(*
SPDX-FileCopyrightText: © 2026 Oleksandr Tiutyk <trofimich@gmail.com>
SPDX-License-Identifier: MIT
License: https://opensource.org/license/mit
*)

(*!
<summary>
Base automation component that coordinates children and routes requests through the component hierarchy.
</summary>
<description>
Action permissions are checked locally and then through parents, stopping at the first rejection. A missing
local policy permits that level; permission is granted only if no level rejects the request. Indexed Try
lookups return borrowed interfaces or null and do not propagate exceptions. Initialization validates required
dependencies before hooks. Each fixed child slot must identify a distinct child whose Parent is this branch.
Cycle-service hooks remain available while disabled in WORKING or STOPPED;
state changes end obsolete child phases. Use one owner task without recursive Execute.
</description>
*)

FUNCTION_BLOCK ABSTRACT BranchAutomationComponent EXTENDS AutomationComponent IMPLEMENTS IParentAutomationComponent
VAR
	{attribute 'hide'} 
	_ActionPermissionPolicy : TOF_Core.IActionPermissionPolicy;
	
	{attribute 'hide'} 
	_ChildCriticalErrorHandlingPolicy : IChildCriticalErrorHandlingPolicy;

	_ChildHierarchyValidated : BOOL;
END_VAR

{attribute 'monitoring' := 'call'}
PROPERTY FINAL ActionPermissionPolicy : TOF_Core.IActionPermissionPolicy
GET
ActionPermissionPolicy := _ActionPermissionPolicy;
END_GET
SET
_ActionPermissionPolicy := ActionPermissionPolicy;
END_SET
END_PROPERTY

METHOD FINAL BroadcastEvent
VAR_INPUT
	event : TOF_Core.IEvent;
END_VAR
VAR
	stopPropagation : BOOL;
	
	i : TOF_Core.INT_INDEX;
	
	child : IChildAutomationComponent;
	childAsBroadcastEventDispatcher : TOF_Core.IBroadcastEventDispatcher;
END_VAR
OnEventReceived(event := event, stopPropagation => stopPropagation);

IF stopPropagation THEN
	RETURN;
END_IF

FOR i := 0 TO ChildCount - 1 DO
	child := TryGetChildByIndex(index := i);
	
	IF child = 0 OR_ELSE NOT __QUERYINTERFACE(child, childAsBroadcastEventDispatcher) THEN
		CONTINUE;
	END_IF
	
	childAsBroadcastEventDispatcher.BroadcastEvent(event := event);
END_FOR
END_METHOD

{attribute 'monitoring' := 'call'}
PROPERTY ABSTRACT ChildCount : TOF_Core.INT_LENGTH
GET
END_GET
END_PROPERTY

{attribute 'monitoring' := 'call'}
PROPERTY FINAL ChildCriticalErrorHandlingPolicy : IChildCriticalErrorHandlingPolicy
GET
ChildCriticalErrorHandlingPolicy := _ChildCriticalErrorHandlingPolicy;
END_GET
SET
_ChildCriticalErrorHandlingPolicy := ChildCriticalErrorHandlingPolicy;
END_SET
END_PROPERTY

(*!
<summary>Disables the branch, its children and invokes disable hooks.</summary>
<description>
Hook or child exceptions propagate to the caller without rolling back already disabled children.
</description>
*)
METHOD FINAL Disable
VAR
	i : INT;
	
	child : IChildAutomationComponent;

	exceptionCode : __SYSTEM.ExceptionCode;
END_VAR
VAR_INST
	disabling : BOOL;
END_VAR
IF NOT _Enabled OR_ELSE disabling THEN
	RETURN;
END_IF

disabling := TRUE;

__TRY
	OnBeforeChildrenDisable();
	
	FOR i := 0 TO ChildCount - 1 DO
		child := TryGetChildByIndex(index := i);
		
		IF child <> 0 THEN
			child.Disable();
		END_IF
	END_FOR
	
	OnAfterChildrenDisable();
	
	_Enabled := FALSE;
	
	disabling := FALSE;	
__CATCH(exceptionCode)
	disabling := FALSE;
	
	TOF_Core.ExceptionManager.ReThrowLastException(
		exceptionCode := exceptionCode,
		catchPointNamespaceName := NamespaceName,
		catchPointPOUName := __POUNAME(),
		catchPointPosition := __POSITION()
	);
__ENDTRY
END_METHOD

(*!
<summary>Advances stopped children while the branch remains enabled and stopped.</summary>
<description>
OnBeforeChildrenStopped may call Reset. A state or enablement change ends this phase before remaining
children or the after-stopped hook. Completed effects remain. Hook failures are logged; other failures may escape.
</description>
*)
METHOD PRIVATE FINAL doStop
VAR
	exceptionCode : __SYSTEM.ExceptionCode;
	exception : TOF_Core.IException;	
	exceptionReaction : TOF_Core.EXCEPTION_REACTION;

	i : INT;
	
	child : IChildAutomationComponent;
END_VAR
__TRY
	OnBeforeChildrenStopped();
__CATCH(exceptionCode)
	exception := TOF_Core.ExceptionManager.GetLastException(
		exceptionCode := exceptionCode,
		catchPointNamespaceName := NamespaceName,
		catchPointPOUName := __POUNAME(),
		catchPointPosition := __POSITION()
	);	

	exceptionReaction := OnHandleException(exception := exception, failedMethodName := 'OnBeforeChildrenStopped');

	TOF_Core.LogManager.TryLogException(
		exception := exception,
		severity := GetErrorSeverityByExceptionReaction(exceptionReaction := exceptionReaction),
		topic1 := "AutomationComponent",
		topic2 := "AutomationComponent.OnBeforeChildrenStopped"
	);
__ENDTRY	

IF NOT Enabled OR_ELSE _OperationalState <> OPERATIONAL_STATE.STOPPED THEN
	RETURN;
END_IF

FOR i := 0 TO ChildCount - 1 DO
	child := TryGetChildByIndex(index := i);
	
	IF child = 0 OR_ELSE NOT child.Enabled THEN
		CONTINUE;
	END_IF
	
	CASE child.OperationalState OF
		OPERATIONAL_STATE.WORKING:			
			child.Stop(reason := TOF_Core.WideStrings.Concat255("Parent device (", Name, ") stopped"));
		
		OPERATIONAL_STATE.STOPPED:
			child.Execute();
	END_CASE

	IF NOT Enabled OR_ELSE _OperationalState <> OPERATIONAL_STATE.STOPPED THEN
		RETURN;
	END_IF
END_FOR

__TRY
	OnAfterChildrenStopped();
__CATCH(exceptionCode)
	exception := TOF_Core.ExceptionManager.GetLastException(
		exceptionCode := exceptionCode,
		catchPointNamespaceName := NamespaceName,
		catchPointPOUName := __POUNAME(),
		catchPointPosition := __POSITION()
	);	

	exceptionReaction := OnHandleException(exception := exception, failedMethodName := 'OnAfterChildrenStopped');

	TOF_Core.LogManager.TryLogException(
		exception := exception,
		severity := GetErrorSeverityByExceptionReaction(exceptionReaction := exceptionReaction),
		topic1 := "AutomationComponent",
		topic2 := "AutomationComponent.OnAfterChildrenStopped"
	);
__ENDTRY
END_METHOD

(*!
<summary>Advances children according to the selected critical-error reaction.</summary>
<description>
Ignore and continue preserve traversal of later children and the after-working hook. Stop ends traversal.
A non-critical error copied from a faulted child under SET_ERROR_AND_CONTINUE is retained without calling
OnRecover while any enabled child still holds a critical error handled with continue. An exception raised by
OnRecover always records a copied CRITICAL error and stops the branch without consulting
ExceptionHandlingPolicy. State or enablement changes end the obsolete phase; completed effects remain.
</description>
*)
METHOD PRIVATE doWork
VAR
	exceptionCode : __SYSTEM.ExceptionCode;
	exception : TOF_Core.IException;	
	exceptionReaction : TOF_Core.EXCEPTION_REACTION;

	childCriticalErrorReaction : CHILD_CRITICAL_ERROR_REACTION;

	i : INT;
	
	child : IChildAutomationComponent;
END_VAR
// automatic non-critical error recovering
IF _OperationalState = OPERATIONAL_STATE.WORKING
	AND_THEN HasError
	AND_THEN _Error.Severity <> TOF_Core.ERROR_SEVERITY.CRITICAL
	AND_THEN NOT hasActiveChildCriticalError()
THEN
	_Error.Clear();
	
	__TRY
		OnRecover();
	__CATCH(exceptionCode)		
		exception := TOF_Core.ExceptionManager.GetLastException(
			exceptionCode := exceptionCode,
			catchPointNamespaceName := NamespaceName,
			catchPointPOUName := __POUNAME(),
			catchPointPosition := __POSITION()
		);

		// An OnRecover failure always stops the branch with a critical error without consulting the policy.
		ProcessException(
			exception := exception,
			exceptionReaction := TOF_Core.EXCEPTION_REACTION.SET_ERROR_AND_STOP,
			exceptionSourceHint := "OnRecover error"
		);

		RETURN;
	__ENDTRY
END_IF

IF NOT Enabled OR_ELSE _OperationalState <> OPERATIONAL_STATE.WORKING THEN
	RETURN;
END_IF

__TRY
	OnBeforeChildrenWorking();
__CATCH(exceptionCode)
	exception := TOF_Core.ExceptionManager.GetLastException(
		exceptionCode := exceptionCode,
		catchPointNamespaceName := NamespaceName,
		catchPointPOUName := __POUNAME(),
		catchPointPosition := __POSITION()
	);	

	exceptionReaction := OnHandleException(exception := exception, failedMethodName := 'OnBeforeChildrenWorking');

	ProcessException(
		exception := exception,
		exceptionReaction := exceptionReaction,
		exceptionSourceHint := "OnBeforeChildrenWorking error"
	);

	IF exceptionReaction = TOF_Core.EXCEPTION_REACTION.SET_ERROR_AND_STOP THEN
		RETURN;		
	END_IF
__ENDTRY	

IF NOT Enabled OR_ELSE _OperationalState <> OPERATIONAL_STATE.WORKING THEN
	RETURN;
END_IF

FOR i := 0 TO ChildCount - 1 DO
	child := TryGetChildByIndex(index := i);
	
	IF child <> 0
		AND_THEN child.Enabled
		AND_THEN (
			child.OperationalState = OPERATIONAL_STATE.WORKING
			OR_ELSE child.OperationalState = OPERATIONAL_STATE.STOPPED
		)
	THEN
		child.Execute();
		
		IF child.HasError AND_THEN child.Error.Severity = TOF_Core.ERROR_SEVERITY.CRITICAL THEN
			childCriticalErrorReaction := HandleChildCriticalError(childWithError := child);
			
			ProcessChildError(
				childError := child.Error,
				childErrorReaction := childCriticalErrorReaction,
				childErrorSourceHint := TOF_Core.WideStrings.Concat255("Child[", TO_WSTRING(i), "](", child.Name, ").Execute error")
			);
			
			IF childCriticalErrorReaction = CHILD_CRITICAL_ERROR_REACTION.SET_ERROR_AND_STOP THEN
				RETURN;
			END_IF
		END_IF
	END_IF

	IF NOT Enabled OR_ELSE _OperationalState <> OPERATIONAL_STATE.WORKING THEN
		RETURN;
	END_IF
END_FOR

__TRY
	OnAfterChildrenWorking();
__CATCH(exceptionCode)
	exception := TOF_Core.ExceptionManager.GetLastException(
		exceptionCode := exceptionCode,
		catchPointNamespaceName := NamespaceName,
		catchPointPOUName := __POUNAME(),
		catchPointPosition := __POSITION()
	);	

	exceptionReaction := OnHandleException(exception := exception, failedMethodName := 'OnAfterChildrenWorking');

	ProcessException(
		exception := exception,
		exceptionReaction := exceptionReaction,
		exceptionSourceHint := "OnAfterChildrenWorking error"
	);

	IF exceptionReaction = TOF_Core.EXCEPTION_REACTION.SET_ERROR_AND_STOP THEN
		RETURN;		
	END_IF
__ENDTRY
END_METHOD

(*!
<summary>Enables the branch, optionally its children, and invokes enable hooks.</summary>
<description>
Enabling does not automatically reset a STOPPED branch or STOPPED children; they remain STOPPED after
Enable until explicitly Reset. If this branch has a disabled parent, enables the parent with
includeChildren := FALSE.
</description>
<param name="includeChildren">When TRUE, recursively enables child components.</param>
*)
METHOD FINAL Enable
VAR_INPUT
	includeChildren : BOOL := TRUE;
END_VAR
VAR
	i : INT;
	
	child : IChildAutomationComponent;

	exceptionCode : __SYSTEM.ExceptionCode;
	
	thisAsChildAutomationComponent : IChildAutomationComponent;
	parent : IParentAutomationComponent;
END_VAR
VAR_INST
	enabling : BOOL;
END_VAR
IF _Enabled OR_ELSE enabling THEN
	RETURN;
END_IF

enabling := TRUE;

__TRY
	OnBeforeChildrenEnable();
	
	IF includeChildren THEN
		FOR i := 0 TO ChildCount - 1 DO
			child := TryGetChildByIndex(index := i);
			
			IF child <> 0 THEN
				child.Enable(includeChildren := includeChildren);
			END_IF
		END_FOR	
	END_IF
	
	OnAfterChildrenEnable();
	
	IF __QUERYINTERFACE(THIS^, thisAsChildAutomationComponent) THEN
		parent := thisAsChildAutomationComponent.Parent;

		IF parent <> 0 AND_THEN NOT parent.Enabled THEN
			parent.Enable(includeChildren := FALSE);
		END_IF
	END_IF
	
	_Enabled := TRUE;
	
	enabling := FALSE;
__CATCH(exceptionCode)
	enabling := FALSE;
	
	TOF_Core.ExceptionManager.ReThrowLastException(
		exceptionCode := exceptionCode,
		catchPointNamespaceName := NamespaceName,
		catchPointPOUName := __POUNAME(),
		catchPointPosition := __POSITION()
	);
__ENDTRY
END_METHOD

(*!
<summary>Services an initialized branch and advances its enabled execution phases.</summary>
<description>
Only WORKING and STOPPED are serviced. Cycle-service hooks run even while disabled, before and after
enabled input, working or stopped, and output phases. They may enable, disable, stop or reset the branch;
enablement is checked again before work and output. INITIALIZING and INVALID do nothing. The final service
hook also follows handled stop reactions; an escaping nested failure may abort the call. Use one owner task
without recursive Execute. Completed callback effects are not rolled back.
</description>
*)
{attribute 'estimated-stack-usage' := '99'}
METHOD FINAL Execute
VAR
	exceptionCode : __SYSTEM.ExceptionCode;
	exception : TOF_Core.IException;
	exceptionReaction : TOF_Core.EXCEPTION_REACTION;
	runEnabledPhases : BOOL;
END_VAR
IF _OperationalState <> OPERATIONAL_STATE.WORKING
	AND_THEN _OperationalState <> OPERATIONAL_STATE.STOPPED
THEN
	RETURN;
END_IF

runEnabledPhases := TRUE;

__TRY
	OnCycleStart();
__CATCH(exceptionCode)
	exception := TOF_Core.ExceptionManager.GetLastException(
		exceptionCode := exceptionCode,
		catchPointNamespaceName := NamespaceName,
		catchPointPOUName := __POUNAME(),
		catchPointPosition := __POSITION()
	);
	exceptionReaction := OnHandleException(exception := exception, failedMethodName := 'OnCycleStart');

	ProcessException(
		exception := exception,
		exceptionReaction := exceptionReaction,
		exceptionSourceHint := "OnCycleStart error"
	);

	IF exceptionReaction = TOF_Core.EXCEPTION_REACTION.SET_ERROR_AND_STOP THEN
		runEnabledPhases := FALSE;
	END_IF
__ENDTRY

IF runEnabledPhases AND_THEN Enabled THEN
	__TRY
		OnBeforeExecute();
	__CATCH(exceptionCode)
		exception := TOF_Core.ExceptionManager.GetLastException(
			exceptionCode := exceptionCode,
			catchPointNamespaceName := NamespaceName,
			catchPointPOUName := __POUNAME(),
			catchPointPosition := __POSITION()
		);
		exceptionReaction := OnHandleException(exception := exception, failedMethodName := 'OnBeforeExecute');

		ProcessException(
			exception := exception,
			exceptionReaction := exceptionReaction,
			exceptionSourceHint := "OnBeforeExecute error"
		);

		IF exceptionReaction = TOF_Core.EXCEPTION_REACTION.SET_ERROR_AND_STOP THEN
			runEnabledPhases := FALSE;
		END_IF
	__ENDTRY

	IF runEnabledPhases AND_THEN Enabled THEN
		CASE _OperationalState OF
			OPERATIONAL_STATE.WORKING:
				doWork();

			OPERATIONAL_STATE.STOPPED:
				doStop();
		END_CASE
	END_IF

	IF runEnabledPhases AND_THEN Enabled THEN
		__TRY
			OnAfterExecute();
		__CATCH(exceptionCode)
			exception := TOF_Core.ExceptionManager.GetLastException(
				exceptionCode := exceptionCode,
				catchPointNamespaceName := NamespaceName,
				catchPointPOUName := __POUNAME(),
				catchPointPosition := __POSITION()
			);
			exceptionReaction := OnHandleException(exception := exception, failedMethodName := 'OnAfterExecute');

			ProcessException(
				exception := exception,
				exceptionReaction := exceptionReaction,
				exceptionSourceHint := "OnAfterExecute error"
			);
		__ENDTRY
	END_IF
END_IF

__TRY
	OnCycleEnd();
__CATCH(exceptionCode)
	exception := TOF_Core.ExceptionManager.GetLastException(
		exceptionCode := exceptionCode,
		catchPointNamespaceName := NamespaceName,
		catchPointPOUName := __POUNAME(),
		catchPointPosition := __POSITION()
	);
	exceptionReaction := OnHandleException(exception := exception, failedMethodName := 'OnCycleEnd');

	ProcessException(
		exception := exception,
		exceptionReaction := exceptionReaction,
		exceptionSourceHint := "OnCycleEnd error"
	);
__ENDTRY
END_METHOD

METHOD GetEffectiveChildCriticalErrorHandlingPolicy : IChildCriticalErrorHandlingPolicy
VAR
	thisAsChildAutomationComponent : IChildAutomationComponent;
	parent : IParentAutomationComponent;
END_VAR
IF _ChildCriticalErrorHandlingPolicy <> 0 THEN
	GetEffectiveChildCriticalErrorHandlingPolicy := _ChildCriticalErrorHandlingPolicy;
ELSIF __QUERYINTERFACE(THIS^, thisAsChildAutomationComponent) THEN
	parent := thisAsChildAutomationComponent.Parent;

	IF parent <> 0 THEN
		GetEffectiveChildCriticalErrorHandlingPolicy := parent.GetEffectiveChildCriticalErrorHandlingPolicy();
	END_IF
END_IF
END_METHOD

METHOD PROTECTED FINAL HandleChildCriticalError : CHILD_CRITICAL_ERROR_REACTION
VAR_INPUT
	childWithError : IChildAutomationComponent;
END_VAR
VAR
	effectiveChildCriticalErrorHandlingPolicy : IChildCriticalErrorHandlingPolicy;
END_VAR
effectiveChildCriticalErrorHandlingPolicy := GetEffectiveChildCriticalErrorHandlingPolicy();

IF effectiveChildCriticalErrorHandlingPolicy <> 0 THEN
	HandleChildCriticalError := effectiveChildCriticalErrorHandlingPolicy.HandleChildCriticalError(
		childWithError := childWithError,
		handlingObject := THIS^
	);
ELSE
	HandleChildCriticalError := CHILD_CRITICAL_ERROR_REACTION.SET_ERROR_AND_STOP;
END_IF
END_METHOD

(*!
<summary>Checks whether any enabled child still holds a critical error handled with continue.</summary>
<description>
Prevents premature automatic non-critical error clearing and OnRecover calls while an enabled child
remains faulted with a critical error under SET_ERROR_AND_CONTINUE.
</description>
*)
METHOD PRIVATE hasActiveChildCriticalError : BOOL
VAR
	i : INT;
	child : IChildAutomationComponent;
	childCriticalErrorReaction : CHILD_CRITICAL_ERROR_REACTION;
END_VAR
FOR i := 0 TO ChildCount - 1 DO
	child := TryGetChildByIndex(index := i);

	IF child <> 0
		AND_THEN child.Enabled
		AND_THEN child.HasError
		AND_THEN child.Error.Severity = TOF_Core.ERROR_SEVERITY.CRITICAL
	THEN
		childCriticalErrorReaction := HandleChildCriticalError(childWithError := child);

		IF childCriticalErrorReaction = CHILD_CRITICAL_ERROR_REACTION.SET_ERROR_AND_CONTINUE THEN
			hasActiveChildCriticalError := TRUE;

			RETURN;
		END_IF
	END_IF
END_FOR
END_METHOD

(*!
<summary>Validates required dependencies and advances branch initialization.</summary>
<description>
Required storage and child slots are checked before initialization hooks. Empty compositions are valid.
Before the first initialization hook, each child must name this branch as Parent and appear in exactly one slot.
Keep the composition stable thereafter. A mismatch or duplicate records a critical error and makes the branch INVALID.
An INVALID child immediately makes this branch INVALID and copies its error when available.
During initialization, the branch expands its effective initialization timeout to at least the maximum
InitializationTimeout of its children. OnAfterChildrenInitializing runs only once all children have completed
initialization. FALSE reports pending work or failure. Caught initialization failures return FALSE and record
a critical error in terminal INVALID. TRUE reports completed initialization, including an already stopped
component. Callback effects are not rolled back. Child types require a live constructor-bound parent.
</description>
*)
METHOD FINAL Initialize : BOOL
VAR
	i : INT;
	previousIndex : INT;
	expectedParent : IParentAutomationComponent;
	childParent : IParentAutomationComponent;
	hierarchyError : WSTRING(255);
		
	child : IChildAutomationComponent;
	previousChild : IChildAutomationComponent;
	childInitialized : BOOL;
	
	exceptionCode : __SYSTEM.ExceptionCode;
	exception : TOF_Core.IException;
	
END_VAR
IF _OperationalState <> OPERATIONAL_STATE.INITIALIZING THEN
	Initialize := _OperationalState <> OPERATIONAL_STATE.INVALID;

	RETURN;
END_IF

__TRY
	Validate();
	expectedParent := THIS^;

	FOR i := 0 TO ChildCount - 1 DO
		child := TryGetChildByIndex(index := i);

		IF child = 0 THEN
			TOF_Core.Exceptions.ThrowDataMemberNotSpecified(
				sourceNamespaceName := NamespaceName,
				sourceClassName := ClassName,
				sourcePOUName := __POUNAME(),
				sourcePosition := __POSITION(),
				dataMemberName := TOF_Core.Strings.Concat255('Child[', TO_STRING(i), ']')
			);			
		END_IF

		IF _ChildHierarchyValidated THEN
			CONTINUE;
		END_IF

		childParent := child.Parent;

		IF childParent <> expectedParent THEN
			hierarchyError := TOF_Core.WideStrings.Concat255(
				Name,
				": Children[",
				TO_WSTRING(i),
				"] (",
				child.Name,
				") has a different Parent"
			);
		ELSE
			FOR previousIndex := 0 TO i - 1 DO
				previousChild := TryGetChildByIndex(index := previousIndex);

				IF previousChild = child THEN
					hierarchyError := TOF_Core.WideStrings.Concat255(
						Name,
						": Children[",
						TO_WSTRING(i),
						"] (",
						child.Name,
						") duplicates Children[",
						TO_WSTRING(previousIndex),
						"]"
					);

					EXIT;
				END_IF
			END_FOR
		END_IF

		IF hierarchyError <> "" THEN
			TOF_Core.Exceptions.ThrowClassInitialization(
				sourceNamespaceName := NamespaceName,
				sourceClassName := ClassName,
				sourcePOUName := __POUNAME(),
				sourcePosition := __POSITION(),
				errorMessage := hierarchyError
			);
		END_IF
	END_FOR

	_ChildHierarchyValidated := TRUE;
	OnBeforeChildrenInitializing();

	IF _InitializationTimer.PT = T#0S THEN
		_InitializationTimer.PT := Parameters.InitializationTimeout;
	END_IF

	Initialize := TRUE;

	FOR i := 0 TO ChildCount - 1 DO
		child := TryGetChildByIndex(index := i);

		IF child = 0 THEN
			TOF_Core.Exceptions.ThrowDataMemberNotSpecified(
				sourceNamespaceName := NamespaceName,
				sourceClassName := ClassName,
				sourcePOUName := __POUNAME(),
				sourcePosition := __POSITION(),
				dataMemberName := TOF_Core.Strings.Concat255('Child[', TO_STRING(i), ']')
			);
		END_IF

		childInitialized := child.Initialize();

		IF child.OperationalState = OPERATIONAL_STATE.INVALID THEN
			Initialize := FALSE;

			IF child.HasError THEN
				_Error := child.Error;
				_Error.SetSeverity(severity := TOF_Core.ERROR_SEVERITY.CRITICAL);
				SetOperationalState(
					state := OPERATIONAL_STATE.INVALID,
					reason := TOF_Core.WideStrings.Concat255("Child[", TO_WSTRING(i), "] initialization failed")
				);

				RETURN;
			END_IF

			TOF_Core.Exceptions.ThrowStandard(
				sourceNamespaceName := NamespaceName,
				sourceClassName := ClassName,
				sourcePOUName := __POUNAME(),
				sourcePosition := __POSITION(),
				message := "A child entered INVALID during initialization without an error diagnostic."
			);
		END_IF

		IF child.InitializationTimeout > _InitializationTimer.PT THEN
			_InitializationTimer.PT := child.InitializationTimeout;
		END_IF

		Initialize := Initialize AND childInitialized;
	END_FOR

	Initialize := Initialize AND_THEN OnAfterChildrenInitializing();
	
	IF Initialize THEN
		SetOperationalState(state := OPERATIONAL_STATE.WORKING, reason := "Successfull initialization");
	ELSE
		_InitializationTimer(IN := TRUE);
		
		IF _InitializationTimer.Q THEN		
			TOF_Core.Exceptions.ThrowTimeout(
				sourceNamespaceName := NamespaceName,
				sourceClassName := ClassName,
				sourcePOUName := __POUNAME(),
				sourcePosition := __POSITION(),
				timeoutValue := _InitializationTimer.PT,
				operationName := "Initialization"
			);
		END_IF		
	END_IF	
__CATCH(exceptionCode)
	Initialize := FALSE;

	IF hierarchyError = "" THEN
		hierarchyError := "Initialization error";
	END_IF

	exception := TOF_Core.ExceptionManager.GetLastException(
		exceptionCode := exceptionCode,
		catchPointNamespaceName := NamespaceName,
		catchPointPOUName := __POUNAME(),
		catchPointPosition := __POSITION()
	);
	
	ProcessException(
		exception := exception,
		exceptionReaction := TOF_Core.EXCEPTION_REACTION.SET_ERROR_AND_CONTINUE,
		exceptionSourceHint := hierarchyError
	);					
__ENDTRY
END_METHOD

METHOD PROTECTED OnAfterChildrenDisable
END_METHOD

METHOD PROTECTED OnAfterChildrenEnable
END_METHOD

(*!
<summary>Completes branch initialization after all children have finished initializing.</summary>
<description>
Invoked only once every child has completed initialization (returned TRUE from Initialize). Return FALSE to
keep the branch in INITIALIZING until a subsequent Initialize call returns TRUE.
</description>
*)
METHOD PROTECTED OnAfterChildrenInitializing : BOOL
OnAfterChildrenInitializing := TRUE;
END_METHOD

METHOD PROTECTED OnAfterChildrenProcessInput
END_METHOD

(*!
<summary>Runs after the branch completes an output pass without changing its operational state.</summary>
<description>Both working and stopped passes may complete. An interrupted pass skips this hook.</description>
*)
METHOD PROTECTED OnAfterChildrenProcessOutput
END_METHOD

METHOD PROTECTED OnAfterChildrenReset
END_METHOD

METHOD PROTECTED OnAfterChildrenStopped
END_METHOD

METHOD PROTECTED OnAfterChildrenWorking
END_METHOD

(*!
<summary>Completes enabled processing after the working or stopped phase.</summary>
<description>
Execute checks Enabled again before calling this hook. STOPPED branches remain eligible. A handled stop
reaction in OnCycleStart or OnBeforeExecute skips this hook. The base implementation does nothing.
Exceptions follow the branch exception policy.
</description>
*)
METHOD PROTECTED OnAfterExecute
END_METHOD

METHOD PROTECTED OnBeforeChildrenDisable
END_METHOD

METHOD PROTECTED OnBeforeChildrenEnable
END_METHOD

(*!
<summary>Runs before child initialization on each pending initialization cycle.</summary>
<description>
Invoked after branch dependencies and child hierarchy validation succeed. Exceptions transition the branch to
terminal INVALID.
</description>
*)
METHOD PROTECTED OnBeforeChildrenInitializing
END_METHOD

METHOD PROTECTED OnBeforeChildrenProcessInput
END_METHOD

METHOD PROTECTED OnBeforeChildrenProcessOutput
END_METHOD

METHOD PROTECTED OnBeforeChildrenReset
END_METHOD

(*!
<summary>Runs before stopped-child traversal.</summary>
<description>
May call Reset. A state or enablement change ends this stopped phase before remaining children
and the after-stopped hook. Do not recursively call Execute.
</description>
*)
METHOD PROTECTED OnBeforeChildrenStopped
END_METHOD

METHOD PROTECTED OnBeforeChildrenWorking
END_METHOD

(*!
<summary>Prepares an enabled branch for its working or stopped phase.</summary>
<description>
Execute calls this hook after OnCycleStart if the branch is enabled and the enabled phases may proceed.
Execute then checks Enabled again and selects the phase using the current operational state. The base
implementation does nothing. Exceptions follow the branch exception policy.
</description>
*)
METHOD PROTECTED OnBeforeExecute
END_METHOD

(*!
<summary>Services the branch after the enabled phases have run or been skipped.</summary>
<description>
Execute reaches this hook even while disabled and after a handled stop reaction. An escaping exception
can end Execute before this hook runs. The base implementation does nothing. Exceptions raised here follow
the branch exception policy.
</description>
*)
METHOD PROTECTED OnCycleEnd
END_METHOD

(*!
<summary>Services the branch before Execute checks Enabled.</summary>
<description>
Execute calls this hook in WORKING and STOPPED, including while disabled. An override can process commands
that enable or disable the branch for this call. The base implementation does nothing. Exceptions follow
the branch exception policy.
</description>
*)
METHOD PROTECTED OnCycleStart
END_METHOD

(*!
<summary>
Checks local permission and then requests permission from the parent, stopping at the first rejection.
</summary>
<description>
A missing local policy permits this level. The local policy receives this branch as evaluatingObject; the
original descriptor and requester are forwarded unchanged to the parent. Returns TRUE only if no level rejects
the request. On FALSE, rejectReason contains the rejecting level's reason; on TRUE it must be ignored.
Evaluation exceptions propagate to the caller without becoming ordinary rejections. Inputs must be non-null
and live. Arguments are borrowed only during this synchronous call, without ownership transfer.
</description>
*)

METHOD FINAL RequestActionPermission : BOOL
VAR_INPUT
	actionDescriptor : TOF_Core.INamed;
	requestingObject : TOF_Core.IObject;
END_VAR
VAR_IN_OUT
	rejectReason : WSTRING(255);
END_VAR
VAR
	thisAsChildAutomationComponent : IChildAutomationComponent;
	parent : IParentAutomationComponent;
END_VAR
IF _ActionPermissionPolicy <> 0 THEN 
	RequestActionPermission := _ActionPermissionPolicy.CheckActionPermission(
		actionDescriptor := actionDescriptor,
		requestingObject := requestingObject,
		evaluatingObject := THIS^,
		rejectReason := rejectReason
	);
ELSE
	RequestActionPermission := TRUE;
END_IF

IF RequestActionPermission
	AND_THEN __QUERYINTERFACE(THIS^, thisAsChildAutomationComponent)
THEN
	parent := thisAsChildAutomationComponent.Parent;

	IF parent <> 0 THEN
		RequestActionPermission := parent.RequestActionPermission(
			actionDescriptor := actionDescriptor,
			requestingObject := requestingObject,
			rejectReason := rejectReason
		);
	END_IF
END_IF
END_METHOD

(*!
<summary>Attempts to resume an enabled stopped branch and its enabled children.</summary>
<description>
Clears the previous branch error before reset hooks. Disabled children are skipped and remain STOPPED if
later enabled until explicitly Reset. A failure of the branch's own reset hook (OnBeforeChildrenReset or
OnAfterChildrenReset) always leaves the branch STOPPED with a copied CRITICAL error without consulting
ExceptionHandlingPolicy; later children are not reset after OnBeforeChildrenReset fails. Ignore and
continue allow later children to reset and the branch to enter WORKING even if a child remains stopped.
Continue copies that error at ERROR severity; ignore leaves it local. Stop leaves the branch STOPPED. Reset
may be called from a stopped-cycle hook, but reset hooks must not reenter Reset. State or enablement changes
end traversal; completed effects remain.
</description>
*)
METHOD FINAL Reset
VAR
	exceptionCode : __SYSTEM.ExceptionCode;
	exception : TOF_Core.IException;	
	
	childCriticalErrorReaction : CHILD_CRITICAL_ERROR_REACTION;
	
	i : INT;
		
	child : IChildAutomationComponent;	
END_VAR
IF NOT Enabled OR_ELSE _OperationalState <> OPERATIONAL_STATE.STOPPED THEN
	RETURN;
END_IF

_Error.Clear();

__TRY
	OnBeforeChildrenReset();
__CATCH(exceptionCode)		
	exception := TOF_Core.ExceptionManager.GetLastException(
		exceptionCode := exceptionCode,
		catchPointNamespaceName := NamespaceName,
		catchPointPOUName := __POUNAME(),
		catchPointPosition := __POSITION()
	);

	// A failed reset hook always keeps the branch STOPPED with a critical error; the policy is not consulted.
	ProcessException(
		exception := exception,
		exceptionReaction := TOF_Core.EXCEPTION_REACTION.SET_ERROR_AND_STOP,
		exceptionSourceHint := "OnBeforeChildrenReset error"
	);

	RETURN;
__ENDTRY

IF NOT Enabled OR_ELSE _OperationalState <> OPERATIONAL_STATE.STOPPED THEN
	RETURN;
END_IF

FOR i := 0 TO ChildCount - 1 DO
	child := TryGetChildByIndex(index := i);
	
	IF child <> 0 AND_THEN child.Enabled THEN
		child.Reset();
		
		IF child.HasError AND_THEN child.Error.Severity = TOF_Core.ERROR_SEVERITY.CRITICAL THEN
			childCriticalErrorReaction := HandleChildCriticalError(childWithError := child);
			
			ProcessChildError(
				childError := child.Error,
				childErrorReaction := childCriticalErrorReaction,
				childErrorSourceHint := TOF_Core.WideStrings.Concat255("Child[", TO_WSTRING(i), "](", child.Name, ").Reset error")
			);

			IF childCriticalErrorReaction = CHILD_CRITICAL_ERROR_REACTION.SET_ERROR_AND_STOP THEN
				RETURN;
			END_IF
		END_IF
	END_IF

	IF NOT Enabled OR_ELSE _OperationalState <> OPERATIONAL_STATE.STOPPED THEN
		RETURN;
	END_IF
END_FOR

__TRY
	OnAfterChildrenReset();
	
	IF Enabled AND_THEN _OperationalState = OPERATIONAL_STATE.STOPPED THEN
		SetOperationalState(state := OPERATIONAL_STATE.WORKING, reason := "Reset");
	END_IF
__CATCH(exceptionCode)		
	exception := TOF_Core.ExceptionManager.GetLastException(
		exceptionCode := exceptionCode,
		catchPointNamespaceName := NamespaceName,
		catchPointPOUName := __POUNAME(),
		catchPointPosition := __POSITION()
	);

	// A failed reset hook always keeps the branch STOPPED with a critical error; the policy is not consulted.
	ProcessException(
		exception := exception,
		exceptionReaction := TOF_Core.EXCEPTION_REACTION.SET_ERROR_AND_STOP,
		exceptionSourceHint := "OnAfterChildrenReset error"
	);
__ENDTRY
END_METHOD

(*!
<summary>Transitions a WORKING branch and all WORKING children to OPERATIONAL_STATE.STOPPED.</summary>
<description>
Stops the branch and all WORKING children regardless of Enabled. Child Stop failures are logged as critical.
</description>
<param name="reason">Descriptive reason stored in OperationalStateReason.</param>
*)
METHOD FINAL Stop
VAR_INPUT
	reason : WSTRING(255) := "External stop";
END_VAR
VAR
	exceptionCode : __SYSTEM.ExceptionCode;
	exception : TOF_Core.IException;	

	i : INT;
	
	child : IChildAutomationComponent;
END_VAR
IF _OperationalState <> OPERATIONAL_STATE.WORKING THEN
	RETURN;
END_IF

SetOperationalState(state := OPERATIONAL_STATE.STOPPED, reason := reason);

FOR i := 0 TO ChildCount - 1 DO
	__TRY
		child := TryGetChildByIndex(index := i); 
		
		IF child <> 0 AND_THEN child.OperationalState = OPERATIONAL_STATE.WORKING THEN		
			child.Stop(reason := TOF_Core.WideStrings.Concat255("Parent (", Name, ") stopped. Reason: ", reason));
		END_IF			
	__CATCH(exceptionCode)
		exception := TOF_Core.ExceptionManager.GetLastException(
			exceptionCode := exceptionCode,
			catchPointNamespaceName := NamespaceName,
			catchPointPOUName := __POUNAME(),
			catchPointPosition := __POSITION()
		);	
		
		TOF_Core.LogManager.TryLogException(
			exception := exception,
			severity := TOF_Core.ERROR_SEVERITY.CRITICAL,
			topic1 := "AutomationComponent",
			topic2 := "AutomationComponent.Stop"
		);
	__ENDTRY
END_FOR
END_METHOD

(*!
<summary>Returns a borrowed child by its zero-based index.</summary>
<description>
Returns null when the entry is unavailable, the index is out of range or a nested call raises an exception.
Fatal allocation observations return null and leave the fatal latch set for the outer task boundary.
Does not transfer ownership or extend lifetime. Implementations must not propagate exceptions.
</description>
*)
METHOD ABSTRACT TryGetChildByIndex : IChildAutomationComponent
VAR_INPUT
	index : TOF_Core.INT_INDEX;
END_VAR
END_METHOD

METHOD PROTECTED ABSTRACT Validate
END_METHOD

END_FUNCTION_BLOCK

(* stored: Version 1.1.0.1
   POU BranchAutomationComponent: Id {179de9c8-6fc8-497c-b86e-77d22d7559c0}, SpecialFunc None
   Folder Methods to override: Id {cd048a51-ca56-4e6a-a6d5-8403d28a5210}
   Folder Cycle: Id {e241a8b9-8315-4b35-90f7-8a965cad1045}
   Folder Disable: Id {130fe9f2-bbd8-4e60-9441-ddfd0141901c}
   Folder Enable: Id {12f5b865-199a-4dd7-8e41-d5e800625ca6}
   Folder Execute: Id {00a453a1-ad8f-47bb-bef6-a6ffcd171789}
   Folder Initialization: Id {d6d336d9-ef91-4b1f-bae4-1c2454b8f6d6}
   Folder ProcessInput: Id {b9bdcde8-d227-4337-a914-5de245b36712}
   Folder ProcessOutput: Id {73c2ab09-04ff-4721-ad1b-e6cc785a336c}
   Folder Reset: Id {7dcb29a2-9973-4885-9f74-1038a5aa2891}
   Folder Stopped: Id {02b22b82-b6c1-49fb-bdb0-d1a9b5d33b8b}
   Folder Working: Id {ece9848d-4500-41ec-adca-c07b101d42a5}
   Folder Service methods: Id {dfdc20d0-90da-4ee2-b28a-a82ad223cd59}
   Property ActionPermissionPolicy: Id {054dbd07-72c3-45f7-894b-093095c1dba6}
   Get Get: Id {07d3e363-d730-4860-822b-273a4c4eec04}
   Set Set: Id {ab25aa7b-2a0e-42ee-aa9e-30c719e242b4}
   Method BroadcastEvent: Id {b3a65959-9192-438d-9b3b-92263d431513}
   Property ChildCount: Id {c2bf4044-8c3f-4694-b502-03d7c6837fdf}
   Get Get: Id {f5f13569-9317-494e-8ad7-d932f7599918}
   Property ChildCriticalErrorHandlingPolicy: Id {3c828eac-4e06-47fc-b519-0e61d3544213}
   Get Get: Id {d119ddbe-a698-4e00-b0b9-ea9b786b87e1}
   Set Set: Id {7450d937-3922-4934-8807-87711ddf39ab}
   Method Disable: Id {9f8a3623-08ea-465f-bfda-4ce58abe2bf9}
   Method doStop: Id {15f6ef78-2e2a-4e13-b736-238af397f6d5}
   Method doWork: Id {1d2f758e-1d18-4c35-861d-3d2b41e9834b}
   Method Enable: Id {b0e28423-49d5-443f-99e6-226254fcb577}
   Method Execute: Id {25cb1f34-284f-498c-958b-8dfda7cade8f}
   Method GetEffectiveChildCriticalErrorHandlingPolicy: Id {55fce35a-19c7-40fd-957d-85f956745e18}
   Method HandleChildCriticalError: Id {839f293e-9205-4a6f-838b-d14dd86be61e}
   Method hasActiveChildCriticalError: Id {f90e4b47-83b5-464a-9e10-913d8591b8f2}
   Method Initialize: Id {24ac7d54-bfdf-430c-8d4e-40b667f55780}
   Method OnAfterChildrenDisable: Id {de10d49d-578e-4a7a-b30d-dcbe7eaa67f7}
   Method OnAfterChildrenEnable: Id {1165a2a7-239a-4bb5-8f3e-e6462d0c1950}
   Method OnAfterChildrenInitializing: Id {6cb14155-7a84-4dd3-a575-77b653934285}
   Method OnAfterChildrenProcessInput: Id {9165bde5-0cf4-4a88-9520-d7dda6cae7ea}
   Method OnAfterChildrenProcessOutput: Id {4df73bdb-052a-4635-a8e1-07d1334a7f95}
   Method OnAfterChildrenReset: Id {862eb02e-c3cf-4f11-b4d0-51cfeec05381}
   Method OnAfterChildrenStopped: Id {70429f04-2ec5-4d13-94eb-bfee5c047e97}
   Method OnAfterChildrenWorking: Id {c97b3a73-c5a9-4482-b28b-882d1d016cd1}
   Method OnAfterExecute: Id {84b329ef-503d-46aa-959d-1e51716064ee}
   Method OnBeforeChildrenDisable: Id {428df434-53b8-4491-9aab-b3a5dd9e3feb}
   Method OnBeforeChildrenEnable: Id {fcc3dec2-5834-4636-9cdd-9eea9043bf97}
   Method OnBeforeChildrenInitializing: Id {3ece4d5d-78d2-4a1b-b7aa-ac08b09e6b07}
   Method OnBeforeChildrenProcessInput: Id {e3339694-bd0c-4309-8526-150debf56b72}
   Method OnBeforeChildrenProcessOutput: Id {baf4b6a4-5565-4d9c-bcf1-5adeadee9802}
   Method OnBeforeChildrenReset: Id {aa65b3fc-dc5d-407d-aeaa-d2722c18b445}
   Method OnBeforeChildrenStopped: Id {0d5d7b0c-eb69-4a7f-b28d-1c85b2de514f}
   Method OnBeforeChildrenWorking: Id {613da739-79e2-4ee2-9175-e0e13072ef84}
   Method OnBeforeExecute: Id {a21a9af0-faff-4c04-9440-53aa1ff069b9}
   Method OnCycleEnd: Id {27d674c2-6f32-44de-ad23-3cb4bd83856e}
   Method OnCycleStart: Id {ce98bb7a-d884-48b6-9057-a833671427c7}
   Method RequestActionPermission: Id {38f3c430-f1b8-4bc0-bb7e-4f38474d7b81}
   Method Reset: Id {0fac72fb-ac13-45be-8a20-c7e96145e4d2}
   Method Stop: Id {da5c54bb-6397-492a-8106-733766e78f84}
   Method TryGetChildByIndex: Id {37f2f3fc-162d-4554-90ba-2cd93bca68c5}
   Method Validate: Id {58f157ed-c4fb-44bd-b2b9-b50da01a7f12} *)
